PROGRAM PRG_Vision

fbMachine.UpdateSlow();

END_PROGRAM

(* stored: Version 1.1.0.1, ProductVersion 3.1.4024.12
   POU PRG_Vision: Id {150307bd-cc4d-4297-ba9b-9aa1f2cc8252}, SpecialFunc None *)
